Staubli VAL3: CartesianSpace.dtx

public pointRx CartesianPos = {fatherId=world[0]}
public num CartesianVel[6]
public num CartesianAccel[6]
public num CartesianForce[6]
public num CarteResVel
public num CarteResAccel
public num CarteResForce
